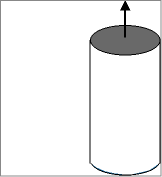
VISUALIZATION VISU_Tube_Top_10  // 162x177
VAR_IN_OUT
	azi : LREAL;
END_VAR
    Ellipse (90,145 70x30)
        p2858320360: azi
    Polygon (90,40) (160,40) (160,162) (155,166) (149,170) (141,172) (132,174) (122,174) (114,173) (105,171) (96,167) (90,162)
        p2858320360: azi
    Ellipse (90,25 70x30)
        p2858320360: azi
    Polygon (120,10) (125,0) (130,10)
        p2858320360: azi
    Polyline (125,37) (125,10)
        p2858320360: azi
    Polyline (90,163) (90,40)
        p2858320360: azi
    Polyline (160,163) (160,40)
        p2858320360: azi
END_VISUALIZATION

(* stored: Version 1.1.0.1, ProductVersion 3.1.4018.5
   Visu VISU_Tube_Top_10: Id {4a459a41-26da-4c8a-963f-ee7c92eac306} *)
